Staubli VAL3: Pallet.pjx

--- Pallet.pjx ---
Parameters version=s7.8.3 stackSize=10000 millimeterUnit=true
Program file=Edit.pgx
Program file=EnterPageKey.pgx
Program file=getFrame.pgx
Program file=getPoint.pgx
Program file=Main.pgx
Program file=MainKey.pgx
Program file=OnF1.pgx
Program file=OnF2.pgx
Program file=OnF7.pgx
Program file=OnF8.pgx
Program file=Refresh.pgx
Program file=RefreshList.pgx
Program file=SetFrame.pgx
Program file=start.pgx
Program file=stop.pgx
Data file=Pallet.dtx
Library alias=user path=Disk://userPage/USERPAGE.pjx
Library alias=Tool path=Disk://Tool/Tool.pjx
Type name=pallet path=Disk://template/pallet/pallet.pjx

--- Pallet.dtx ---
bool bExit
bool bListRefresh
bool bUserRefresh
public frame fFrame = {fatherId=world[0]}
mdesc mNomSpeed
num nPage = 1
num nSelected
num nType
public pallet uPallet{}
  [pallet1]
    frame fFrame
    num ndX
    num ndY
    pointRx pO = {x=493.537278, y=141.157682, z=-16.022447, rx=-172.031241, ry=0.156426, rz=65.99326, shoulder=lefty, elbow=epositive, wrist=wpositive, fatherId=world[0]}
    pointRx pStart
    pointRx pX
    pointRx pY
    string sToolName = "tool6"
  [pallet2]
    frame fFrame
    num ndX
    num ndY
    pointRx pO = {x=493.537278, y=141.157682, z=-16.022447, rx=-172.031241, ry=0.156426, rz=65.99326, shoulder=lefty, elbow=epositive, wrist=wpositive, fatherId=world[0]}
    pointRx pStart
    pointRx pX
    pointRx pY
    string sToolName
pointRx pPonit[3]
  [0] = {x=493.537278, y=141.157682, z=-16.022447, rx=-172.031241, ry=0.156426, rz=65.99326, fatherId=world[0]}
  [1] = {fatherId=world[0]}
  [2] = {fatherId=world[0]}
string sFrameName
string sItem = "pallet1"
string sList[2]
  [0] = "pallet1"
  [1] = "pallet2"
string sListItemValue[7]
  [3] = "0    "
  [4] = "0    "
  [6] = "tool6"
string sParameter[7]
  [0] = "原点     :          "
  [1] = "X点      :          "
  [2] = "Y点      :          "
  [3] = "dX       :0         "
  [4] = "dY       :0         "
  [5] = "起点     :          "
  [6] = "工具     :tool6     "
tool tTool = {fatherId=flange[0], ioLink=valve1}

--- Main.pgx ---
public program Main(num x_nType (dimensions=1))
  local num l_nKey
begin
  //
  bUserRefresh=bListRefresh=true
  bExit=false
  nType=x_nType
  nPage=0
  //
  do
    call Refresh()
    call RefreshList()
    call user:setList("码盘",sList,bUserRefresh,bListRefresh,nSelected,sItem,l_nKey)
    bUserRefresh=false
    bListRefresh=false
    call MainKey(l_nKey)
    delay(0)
  until bExit

end

--- start.pgx ---
public program start()
begin
  call Main(0)
end

--- Edit.pgx ---
program Edit(string x_sName)
  local bool l_bRes
  local num l_i
  local num l_nKey
  local num l_nRes
  local num l_nSelect
  local string l_sItem
  local string l_sValue
begin
  //edit the pallet
  cls()
  resize(sParameter,1,7)
  sParameter[0]="原点"
  sParameter[1]="X点"
  sParameter[2]="Y点"
  sParameter[3]="dX"
  sParameter[4]="dY"
  sParameter[5]="起点"
  sParameter[6]="工具"
  //
  resize(sListItemValue,1,size(sParameter))
  sListItemValue[0]=""
  sListItemValue[1]=""
  sListItemValue[2]=""
  sListItemValue[3]=toString(".3",uPallet[x_sName].ndX)
  sListItemValue[4]=toString(".3",uPallet[x_sName].ndY)
  sListItemValue[5]=""
  sListItemValue[6]=uPallet[sItem].sToolName

  //
  for l_i=0 to size(sParameter)-1
    call user:strlength(sParameter[l_i],user:nBottomX/2)
    l_sValue=sListItemValue[l_i]
    call user:strlength(l_sValue,user:nBottomX/2+1)
    sParameter[l_i]=sParameter[l_i]+":"+l_sValue
  endFor

  bUserRefresh=true
  bListRefresh=true
  nPage=1
  pPonit[0].trsf=uPallet[sItem].pO.trsf
  pPonit[1].trsf=uPallet[sItem].pX.trsf
  pPonit[2].trsf=uPallet[sItem].pY.trsf
  //
  do
    call Refresh()
    call user:setList(x_sName,sParameter,bUserRefresh,bListRefresh,nSelected,l_sItem,l_nKey)
    bUserRefresh=false
    bListRefresh=false
    call EnterPageKey(l_nKey,nSelected,sParameter[nSelected])
    delay(0)
  until l_nKey==255 or l_nKey==278
  //保存坐标系
  pPonit[0].trsf=uPallet[sItem].pO.trsf
  pPonit[1].trsf=uPallet[sItem].pX.trsf
  pPonit[2].trsf=uPallet[sItem].pY.trsf
  setFrame(pPonit[0],pPonit[1],pPonit[2],fFrame)
  //
  libSave()
  nPage=0
  bUserRefresh=true
  bListRefresh=true
end

--- EnterPageKey.pgx ---
program EnterPageKey(num& x_nKey, num& x_nSelect, string& x_sItem)
  local bool l_bRes
  local num l_nItem
  local num l_nKey
  local num l_nView
  local string l_sEmpty
  local string l_sItem
  local string l_sStr
  local string l_sTool
  local string l_sValue
  local string l_sYN[2]
  local point lp
begin
  //
  switch x_nSelect
    case 0
      if x_nKey==271
        uPallet[sItem].pO=here(tTool,world)
        popUpMsg("OK")
      endIf

    break
    case 1
      if x_nKey==271
        uPallet[sItem].pO=here(tTool,world)
        popUpMsg("OK")
      endIf

    break
    case 2
      if x_nKey==271
        uPallet[sItem].pO=here(tTool,world)
        popUpMsg("OK")
      endIf

    break

    case 3
      if x_nKey==270
        call user:editNum(x_sItem,sListItemValue[x_nSelect],uPallet[sItem].ndX,x_nSelect)
      endIf
    break
    case 4
      if x_nKey==270
        call user:editNum(x_sItem,sListItemValue[x_nSelect],uPallet[sItem].ndY,x_nSelect)
      endIf
    break

    case 5
      if x_nKey==271
        if setFrame(pPonit[0],pPonit[1],pPonit[2],fFrame)==0
          uPallet[sItem].pStart=here(tTool,fFrame)
          popUpMsg("OK")
        else
          uPallet[sItem].pStart=here(tTool,fFrame)
          popUpMsg("请先记录原点，X点和Y点！")
        endIf
      endIf
    break

  endSwitch
  //
  if x_nKey==272
    call Tool:Main(1)
    call Tool:getTool(l_sTool,tTool)
    if l_sTool!=""
      uPallet[sItem].sToolName=l_sTool
      sParameter[6]="工具"
      sListItemValue[6]=uPallet[sItem].sToolName
      call user:strlength(sParameter[6],user:nBottomX/2)
      l_sValue=sListItemValue[6]
      call user:strlength(l_sValue,user:nBottomX/2+1)
      sParameter[6]=sParameter[6]+":"+l_sValue
    endIf
    if x_nKey==270 or x_nKey==272
      bUserRefresh=true
      bListRefresh=true
    endIf
  endIf

end

--- getFrame.pgx ---
public program getFrame(string& x_sFrm (dimensions=1))
begin
  x_sFrm=sFrameName

end

--- getPoint.pgx ---
public program getPoint(trsf& x_trPoint, string x_sPallet)
begin
end

--- MainKey.pgx ---
program MainKey(num x_nKey (dimensions=1))
  local num l_nKey
begin
  //
  switch x_nKey
    //
    case 271
      call OnF1()
    break
    //编辑
    case 272
      call OnF2()
    break
    //
    case 273
      //call OnF3()
    break
    //
    case 274
      // call OnF4()
    break
    //
    case 275
    break
    //
    case 276
      //call OnF6()
    break
    //save
    case 277
      call OnF7()
    break
    //返回
    case 278
      call OnF8("是否返回")
    break

  endSwitch
end

--- OnF1.pgx ---
program OnF1()
begin
  switch nPage
    case 0
      call Edit(sItem)
    break
    case 1
      switch nSelected
        case 0
          uPallet[sItem].pO=here(tTool,world)
          popUpMsg("OK")
        break
        case 1
          uPallet[sItem].pO=here(tTool,world)
          popUpMsg("OK")
        break
        case 2
          uPallet[sItem].pO=here(tTool,world)
          popUpMsg("OK")
        break
      endSwitch
    break

  endSwitch
end

--- OnF2.pgx ---
program OnF2()
begin

end

--- OnF7.pgx ---
program OnF7()
begin
  //
  libSave()
  popUpMsg("保存完毕!")
end

--- Refresh.pgx ---
program Refresh()
begin
  //
  if bUserRefresh
    cls()
    userPage()
    switch nPage
      case 0
        gotoxy(1,1)
        put("F1->编辑")
        gotoxy(1,13)
        put("F1")

        //      gotoxy(1,2)
        //      put("F2->工具")
        //      gotoxy(6,13)
        //      put("F2")
        //    gotoxy(1,3)
        //    put("F3->删除")
        //    gotoxy(11,13)
        //    put("F3")
        //    gotoxy(1,4)
        //    put("F4->编辑路径")
        //    gotoxy(16,13)
        //    put("编辑")
        //
        //    gotoxy(1,6)
        //    put("F6->")
        //    gotoxy(26,13)
        //    put("")
        //      gotoxy(1,7)
        //      put("F7->保存")
        //      gotoxy(31,13)
        //      put("F7")
        gotoxy(1,8)
        put("F8->返回")
        gotoxy(36,13)
        put("F8")
      break
      case 1
        gotoxy(1,1)
        put("F1->记录位置")
        gotoxy(1,13)
        put("F1")

        gotoxy(1,2)
        put("F2->工具")
        gotoxy(6,13)
        put("F2")
        //    gotoxy(1,3)
        //    put("F3->删除")
        //    gotoxy(11,13)
        //    put("F3")
        //    gotoxy(1,4)
        //    put("F4->编辑路径")
        //    gotoxy(16,13)
        //    put("编辑")
        //
        //    gotoxy(1,6)
        //    put("F6->")
        //    gotoxy(26,13)
        //    put("")
        //      gotoxy(1,7)
        //      put("F7->保存")
        //      gotoxy(31,13)
        //      put("F7")
        gotoxy(1,8)
        put("F8->返回")
        gotoxy(36,13)
        put("F8")

      break
    endSwitch
  endIf
end

--- RefreshList.pgx ---
program RefreshList()
  local num l_ni
begin
  //
  if bListRefresh
    switch nPage
      case 0
        resize(sList,1,2)
        for l_ni=0 to 1
          sList[l_ni]="pallet"+toString("",l_ni+1)
        endFor
      break

      case 1

      break
    endSwitch
  endIf

end

--- SetFrame.pgx ---
public program SetFrame(string x_sFrame (dimensions=1))
begin
  //
  sFrameName=x_sFrame
end
